// TIA Portal V18 export
FUNCTION_BLOCK "MaterialGate"   // FB5210, LAD
{ S7_Optimized_Access := 'FALSE' }
VERSION : 0.1
// stored: AutoNumber false, IsIECCheckEnabled false, SetENOAutomatically false, UDAEnableTagReadback false
   VAR_INPUT
      iSysInface : "RCS_SysComInterface_V1";
      "iMaterialGate Opened Monitor" : Bool;   // 安全门打开状态监控
      "iMaterialGate Locked Monitor" : Bool;   // 安全门锁定状态监控
      i1s_Pulse : Bool;   // 1s脉冲信号
      "iMaterialGate AutoLock Timer" : Time := T#1s;   // 安全门自动模式下锁延时
      "iMaterialGate ManualLock Timer" : Time := T#60s;   // 安全门手动模式下锁定延时
   END_VAR
   VAR_OUTPUT
      "oMaterialGate LockedLamp" { ExternalAccessible := 'False'; ExternalVisible := 'False'; ExternalWritable := 'False'} : Bool;   // 安全门解锁输出状态
   END_VAR
   VAR_IN_OUT
      ioMaterialGateLock : Bool;   // 安全门锁定输出
      ioHMI_Interface : "SafetyGateUDT";
   END_VAR
   VAR DB_SPECIFIC
      "sMaterialafetyGate Timer" { S7_SetPoint := 'True'} : Array[1..5] of TON_TIME;
      sP_Trig : Array[1..10] of Bool;
      sN_Trig : Array[1..10] of Bool;
      "sMaterialGate UnlockRequest" { ExternalAccessible := 'False'; ExternalVisible := 'False'; ExternalWritable := 'False'} : Bool;   // 安全门开门请求标志位
      "sMaterialGate LockRequest" : Bool;
   END_VAR
   VAR_TEMP
      tAlyways_On : Bool;
      tAlyways_Off : Bool;
   END_VAR
   VAR_TEMP   // added for the SCL form of the ladder/FBD networks
      _w1 : Bool;
      _w2 : Bool;
      _w3 : Bool;
      _w4 : Bool;
      _w5 : Bool;
      _w6 : Bool;
      _w7 : Bool;
   END_VAR
BEGIN

REGION Network 1: #tAlyways_On
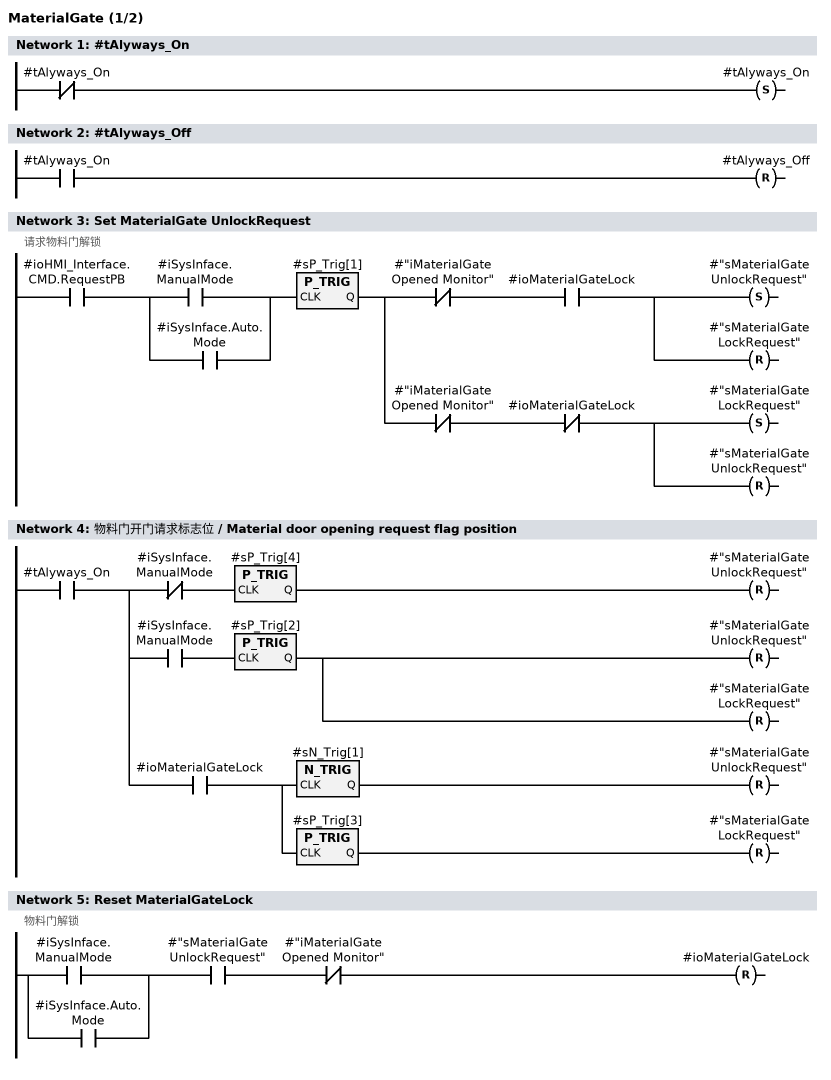
   RUNG wire#powerrail
      I_Contact( #tAlyways_On )
      S_Coil( #tAlyways_On )
   END_RUNG
   // the same network as SCL:
   IF NOT #tAlyways_On THEN #tAlyways_On := TRUE; END_IF;
END_REGION

REGION Network 2: #tAlyways_Off
   RUNG wire#powerrail
      Contact( #tAlyways_On )
      R_Coil( #tAlyways_Off )
   END_RUNG
   // the same network as SCL:
   IF #tAlyways_On THEN #tAlyways_Off := FALSE; END_IF;
END_REGION

REGION Network 3: Set MaterialGate UnlockRequest
   // 请求物料门解锁
   RUNG wire#powerrail
      Contact( #ioHMI_Interface.CMD.RequestPB )
      wire#w1
      Contact( #iSysInface.ManualMode )
      wire#w2
      P_Trig( #sP_Trig[1] )
      wire#w3
      I_Contact( #"iMaterialGate Opened Monitor" )
      Contact( #ioMaterialGateLock )
      wire#w4
      S_Coil( #"sMaterialGate UnlockRequest" )
   END_RUNG
   RUNG wire#w1
      Contact( #iSysInface.Auto.Mode )
   END_RUNG wire#w2
   RUNG wire#w4
      R_Coil( #"sMaterialGate LockRequest" )
   END_RUNG
   RUNG wire#w3
      I_Contact( #"iMaterialGate Opened Monitor" )
      I_Contact( #ioMaterialGateLock )
      wire#w5
      S_Coil( #"sMaterialGate LockRequest" )
   END_RUNG
   RUNG wire#w5
      R_Coil( #"sMaterialGate UnlockRequest" )
   END_RUNG
   // the same network as SCL:
   #_w1 := #ioHMI_Interface.CMD.RequestPB AND (#iSysInface.ManualMode OR #iSysInface.Auto.Mode);
   #_w2 := #_w1 AND NOT #sP_Trig[1];   // rising edge
   #sP_Trig[1] := #_w1;
   IF #_w2 AND NOT #"iMaterialGate Opened Monitor" AND #ioMaterialGateLock THEN
       #"sMaterialGate UnlockRequest" := TRUE;
       #"sMaterialGate LockRequest" := FALSE;
   END_IF;
   IF #_w2 AND NOT #"iMaterialGate Opened Monitor" AND NOT #ioMaterialGateLock THEN
       #"sMaterialGate LockRequest" := TRUE;
       #"sMaterialGate UnlockRequest" := FALSE;
   END_IF;
END_REGION

REGION Network 4: 物料门开门请求标志位 / Material door opening request flag position
   RUNG wire#powerrail
      Contact( #tAlyways_On )
      wire#w1
      I_Contact( #iSysInface.ManualMode )
      P_Trig( #sP_Trig[4] )
      R_Coil( #"sMaterialGate UnlockRequest" )
   END_RUNG
   RUNG wire#w1
      Contact( #iSysInface.ManualMode )
      P_Trig( #sP_Trig[2] )
      wire#w2
      R_Coil( #"sMaterialGate UnlockRequest" )
   END_RUNG
   RUNG wire#w2
      R_Coil( #"sMaterialGate LockRequest" )
   END_RUNG
   RUNG wire#w1
      Contact( #ioMaterialGateLock )
      wire#w3
      N_Trig( #sN_Trig[1] )
      R_Coil( #"sMaterialGate UnlockRequest" )
   END_RUNG
   RUNG wire#w3
      P_Trig( #sP_Trig[3] )
      R_Coil( #"sMaterialGate LockRequest" )
   END_RUNG
   // the same network as SCL:
   #_w1 := #tAlyways_On AND NOT #iSysInface.ManualMode;
   #_w2 := #_w1 AND NOT #sP_Trig[4];   // rising edge
   #sP_Trig[4] := #_w1;
   IF #_w2 THEN #"sMaterialGate UnlockRequest" := FALSE; END_IF;
   #_w3 := #tAlyways_On AND #iSysInface.ManualMode;
   #_w4 := #_w3 AND NOT #sP_Trig[2];   // rising edge
   #sP_Trig[2] := #_w3;
   IF #_w4 THEN
       #"sMaterialGate UnlockRequest" := FALSE;
       #"sMaterialGate LockRequest" := FALSE;
   END_IF;
   #_w5 := #tAlyways_On AND #ioMaterialGateLock;
   #_w6 := NOT #_w5 AND #sN_Trig[1];   // falling edge
   #sN_Trig[1] := #_w5;
   IF #_w6 THEN #"sMaterialGate UnlockRequest" := FALSE; END_IF;
   #_w7 := #_w5 AND NOT #sP_Trig[3];   // rising edge
   #sP_Trig[3] := #_w5;
   IF #_w7 THEN #"sMaterialGate LockRequest" := FALSE; END_IF;
END_REGION

REGION Network 5: Reset MaterialGateLock
   // 物料门解锁
   RUNG wire#powerrail
      Contact( #iSysInface.ManualMode )
      wire#w1
      Contact( #"sMaterialGate UnlockRequest" )
      I_Contact( #"iMaterialGate Opened Monitor" )
      R_Coil( #ioMaterialGateLock )
   END_RUNG
   RUNG wire#powerrail
      Contact( #iSysInface.Auto.Mode )
   END_RUNG wire#w1
   // the same network as SCL:
   IF (#iSysInface.ManualMode OR #iSysInface.Auto.Mode) AND #"sMaterialGate UnlockRequest" AND NOT #"iMaterialGate Opened Monitor" THEN
       #ioMaterialGateLock := FALSE;
   END_IF;
END_REGION

REGION Network 6: Set MaterialGate Lock
   // 物料门锁定
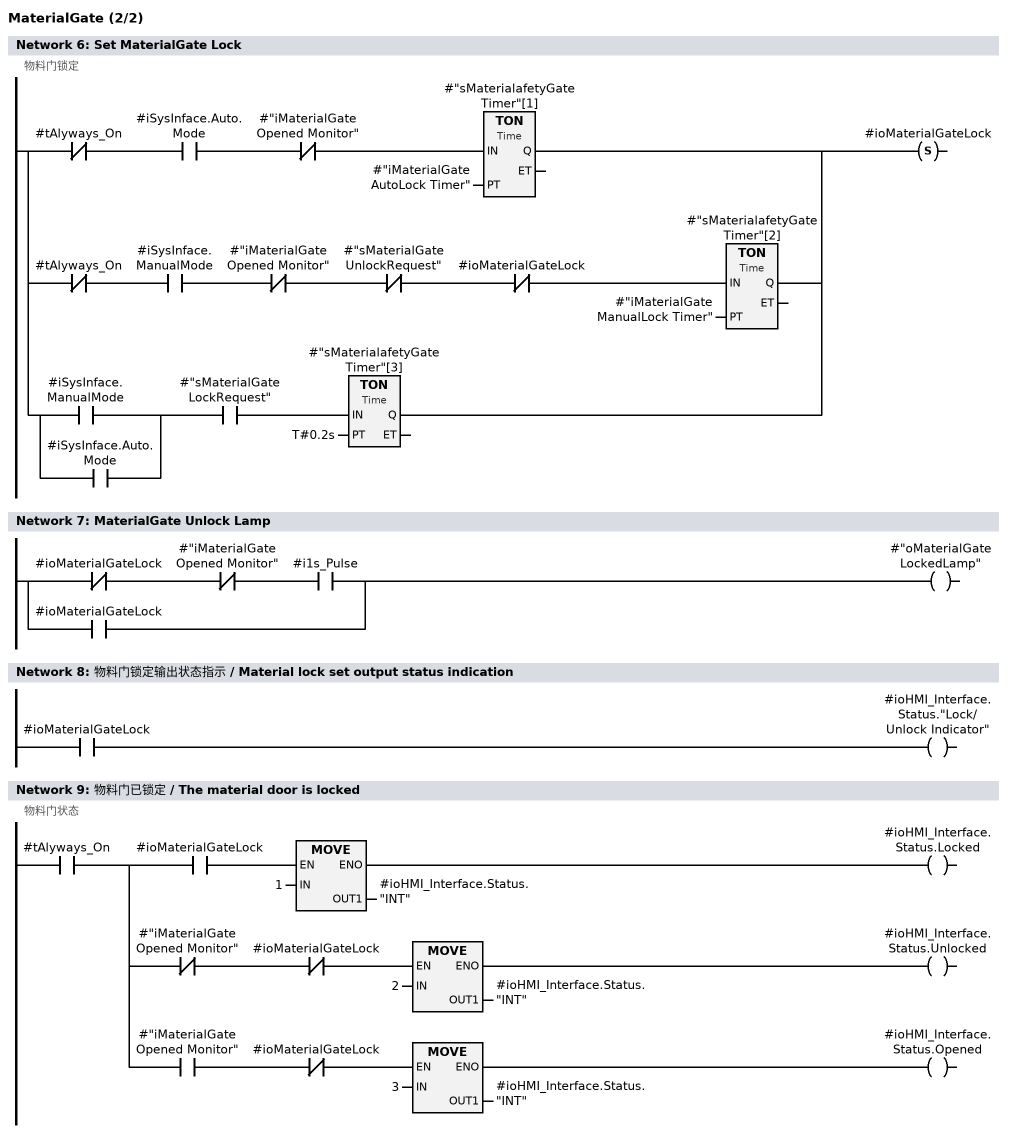
   RUNG wire#powerrail
      I_Contact( #tAlyways_On )
      Contact( #iSysInface.Auto.Mode )
      I_Contact( #"iMaterialGate Opened Monitor" )
      { S7_Templates := "time_type := Time" } #"sMaterialafetyGate Timer"[1].TON(pt := #"iMaterialGate AutoLock Timer", et =>)
      wire#w1
      S_Coil( #ioMaterialGateLock )
   END_RUNG
   RUNG wire#powerrail
      I_Contact( #tAlyways_On )
      Contact( #iSysInface.ManualMode )
      I_Contact( #"iMaterialGate Opened Monitor" )
      I_Contact( #"sMaterialGate UnlockRequest" )
      I_Contact( #ioMaterialGateLock )
      { S7_Templates := "time_type := Time" } #"sMaterialafetyGate Timer"[2].TON(pt := #"iMaterialGate ManualLock Timer", et =>)
   END_RUNG wire#w1
   RUNG wire#powerrail
      Contact( #iSysInface.ManualMode )
      wire#w2
      Contact( #"sMaterialGate LockRequest" )
      { S7_Templates := "time_type := Time" } #"sMaterialafetyGate Timer"[3].TON(pt := T#0.2s, et =>)
   END_RUNG wire#w1
   RUNG wire#powerrail
      Contact( #iSysInface.Auto.Mode )
   END_RUNG wire#w2
   // the same network as SCL:
   #"sMaterialafetyGate Timer"[1].TON(IN := NOT #tAlyways_On AND #iSysInface.Auto.Mode AND NOT #"iMaterialGate Opened Monitor",
                           PT := #"iMaterialGate AutoLock Timer");
   #_w1 := #"sMaterialafetyGate Timer"[1].Q;
   #"sMaterialafetyGate Timer"[2].TON(IN := NOT #tAlyways_On AND #iSysInface.ManualMode AND NOT #"iMaterialGate Opened Monitor" AND NOT #"sMaterialGate UnlockRequest" AND NOT #ioMaterialGateLock,
                           PT := #"iMaterialGate ManualLock Timer");
   #_w2 := #"sMaterialafetyGate Timer"[2].Q;
   #"sMaterialafetyGate Timer"[3].TON(IN := (#iSysInface.ManualMode OR #iSysInface.Auto.Mode) AND #"sMaterialGate LockRequest",
                           PT := T#0.2s);
   IF #_w1 OR #_w2 OR #"sMaterialafetyGate Timer"[3].Q THEN #ioMaterialGateLock := TRUE; END_IF;
END_REGION

REGION Network 7: MaterialGate Unlock Lamp
   RUNG wire#powerrail
      I_Contact( #ioMaterialGateLock )
      I_Contact( #"iMaterialGate Opened Monitor" )
      Contact( #i1s_Pulse )
      wire#w1
      Coil( #"oMaterialGate LockedLamp" )
   END_RUNG
   RUNG wire#powerrail
      Contact( #ioMaterialGateLock )
   END_RUNG wire#w1
   // the same network as SCL:
   #"oMaterialGate LockedLamp" := (NOT #ioMaterialGateLock AND NOT #"iMaterialGate Opened Monitor" AND #i1s_Pulse) OR #ioMaterialGateLock;
END_REGION

REGION Network 8: 物料门锁定输出状态指示 / Material lock set output status indication
   RUNG wire#powerrail
      Contact( #ioMaterialGateLock )
      Coil( #ioHMI_Interface.Status."Lock/Unlock Indicator" )
   END_RUNG
   // the same network as SCL:
   #ioHMI_Interface.Status."Lock/Unlock Indicator" := #ioMaterialGateLock;
END_REGION

REGION Network 9: 物料门已锁定 / The material door is locked
   // 物料门状态
   RUNG wire#powerrail
      Contact( #tAlyways_On )
      wire#w1
      Contact( #ioMaterialGateLock )
      Move(in := 1, out1 => #ioHMI_Interface.Status."INT")
      Coil( #ioHMI_Interface.Status.Locked )
   END_RUNG
   RUNG wire#w1
      I_Contact( #"iMaterialGate Opened Monitor" )
      I_Contact( #ioMaterialGateLock )
      Move(in := 2, out1 => #ioHMI_Interface.Status."INT")
      Coil( #ioHMI_Interface.Status.Unlocked )
   END_RUNG
   RUNG wire#w1
      Contact( #"iMaterialGate Opened Monitor" )
      I_Contact( #ioMaterialGateLock )
      Move(in := 3, out1 => #ioHMI_Interface.Status."INT")
      Coil( #ioHMI_Interface.Status.Opened )
   END_RUNG
   // the same network as SCL:
   #_w1 := #tAlyways_On AND #ioMaterialGateLock;
   IF #_w1 THEN #ioHMI_Interface.Status."INT" := 1; END_IF;
   #ioHMI_Interface.Status.Locked := #_w1;
   #_w2 := #tAlyways_On AND NOT #"iMaterialGate Opened Monitor" AND NOT #ioMaterialGateLock;
   IF #_w2 THEN #ioHMI_Interface.Status."INT" := 2; END_IF;
   #ioHMI_Interface.Status.Unlocked := #_w2;
   #_w3 := #tAlyways_On AND #"iMaterialGate Opened Monitor" AND NOT #ioMaterialGateLock;
   IF #_w3 THEN #ioHMI_Interface.Status."INT" := 3; END_IF;
   #ioHMI_Interface.Status.Opened := #_w3;
END_REGION
END_FUNCTION_BLOCK
